// TIA Portal V16 export
// export: Created 2021-11-12T13:32:33.1039657Z, ExportSetting WithDefaults, DisplayName Totally Integrated Automation Portal, DisplayVersion V16 Update 3, DisplayName TIA Portal Version Control Interface, DisplayVersion V16 Update 2, DisplayName TIA Portal Openness, DisplayVersion V16 Update 3, DisplayName SINAMICS Startdrive Advanced, DisplayVersion V16 Update 5, DisplayName SINAMICS Startdrive G130, G150, S120, S150, SINAMICS MV, S210, DisplayVersion V16 Update 5, DisplayName SINAMICS Startdrive G110M, G120, G120C, G120D, G120P, G115D, DisplayVersion V16 Update 5, DisplayName STEP 7 Professional, DisplayVersion V16 Update 3, DisplayName STEP 7 Safety, DisplayVersion V16, DisplayName WinCC UA Professional, DisplayVersion V16 Update 3
DATA_BLOCK "HMI_PARAM_Zone100"   // DB19
{ S7_Optimized_Access := 'TRUE'; DB_Accessible_From_OPC_UA := 'FALSE' }
VERSION : 0.1
// stored: AutoNumber true, DBAccessibleFromOPCUA false, IsOnlyStoredInLoadMemory false, IsRetainMemResEnabled false, IsWriteProtectedInAS false, MemoryReserve 100
   VAR
      Mode : "UDT_Zone_Parameter";   // Parameters of zone 100
      StationKAS1_Mode : "UDT_Station_Parameter";   // Parameters of station saw KAS1
      StationKAS2_Mode { S7_SetPoint := 'True'} : "UDT_Station_Parameter";   // Parameters of station saw KAS2
      Station110_Mode { S7_SetPoint := 'True'} : "UDT_Station_Parameter";   // Parameters of station 110
      Station120_Mode { S7_SetPoint := 'True'} : "UDT_Station_Parameter";   // Parameters of station 120
      Station1R1_Mode { S7_SetPoint := 'True'} : "UDT_Station_Parameter";   // Parameters of station 1R1
      Station1R2_Mode { S7_SetPoint := 'True'} : "UDT_Station_Parameter";   // Parameters of station 1R2
      Station130_Mode { S7_SetPoint := 'True'} : "UDT_Station_Parameter";   // Parameters of station 130
      Station140_Mode { S7_SetPoint := 'True'} : "UDT_Station_Parameter";   // Parameters of station 140
      Station1R3_Mode { S7_SetPoint := 'True'} : "UDT_Station_Parameter";   // Parameters of station 1R3
      Station1R4_Mode { S7_SetPoint := 'True'} : "UDT_Station_Parameter";   // Parameters of station 1R4
      Station150_Mode { S7_SetPoint := 'True'} : "UDT_Station_Parameter";   // Parameters of station 150
      Station160_Mode { S7_SetPoint := 'True'} : "UDT_Station_Parameter";   // Parameters of station 160
      Station170_Mode { S7_SetPoint := 'True'} : "UDT_Station_Parameter";   // Parameters of station 170
      Station180_Mode { S7_SetPoint := 'True'} : "UDT_Station_Parameter";   // Parameters of station 180
      Station1R5_Mode { S7_SetPoint := 'True'} : "UDT_Station_Parameter";   // Parameters of station 1R5
      Station1R6_Mode { S7_SetPoint := 'True'} : "UDT_Station_Parameter";   // Parameters of station 1R6
      StationBSN1_Mode { S7_SetPoint := 'True'} : "UDT_Station_Parameter";   // Parameters of station furnace BSN1
      StationBSN2_Mode { S7_SetPoint := 'True'} : "UDT_Station_Parameter";   // Parameters of station furnace BSN2
      xxxxx___Alarms___xxxxx { S7_SetPoint := 'True'} : Byte;
      "UF01-SF01_ES" : "UDT_DI_Mon_Parameter";   // E-stop 100UF01-SF01
      QQ01_ES { S7_SetPoint := 'True'} : "UDT_DI_Mon_Parameter";   // E-stop gate 100QQ01
      QQ02_ES { S7_SetPoint := 'True'} : "UDT_DI_Mon_Parameter";   // E-stop gate 100QQ02
      QQ03_ES { S7_SetPoint := 'True'} : "UDT_DI_Mon_Parameter";   // E-stop gate 100QQ03
      QQ04_ES { S7_SetPoint := 'True'} : "UDT_DI_Mon_Parameter";   // E-stop gate 100QQ04
      QQ05_ES { S7_SetPoint := 'True'} : "UDT_DI_Mon_Parameter";   // E-stop gate 100QQ05
      QQ06_ES { S7_SetPoint := 'True'} : "UDT_DI_Mon_Parameter";   // E-stop gate 100QQ06
      QQ07_ES { S7_SetPoint := 'True'} : "UDT_DI_Mon_Parameter";   // E-stop gate 100QQ07
      QQ08_ES { S7_SetPoint := 'True'} : "UDT_DI_Mon_Parameter";   // E-stop gate 100QQ08
      "RU01-KF01" { S7_SetPoint := 'True'} : "UDT_DI_Mon_Parameter";   // gate module 100RU01-KF01
      "RU01-KF02" { S7_SetPoint := 'True'} : "UDT_DI_Mon_Parameter";   // gate module 100RU01-KF01
      "RU01-KF03" { S7_SetPoint := 'True'} : "UDT_DI_Mon_Parameter";   // gate module 100RU01-KF01
   END_VAR
BEGIN
   Mode.HMI1.FuncBtnPanelNr := 10;
   Mode.HMI2.FuncBtnPanelNr := 20;
   Mode.HMI3.FuncBtnPanelNr := 30;
END_DATA_BLOCK
